SUBAPPLICATION Sitzventile (* Subapplication Type *)
  (* Standard: 61499-2 *)
  (* Version 1.0, 2023-02-11, franz *)
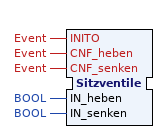
  EVENT_INPUT
    INITO;
    CNF_heben;
    CNF_senken;
  END_EVENT
  VAR_INPUT
    IN_heben : BOOL;
    IN_senken : BOOL;
  END_VAR
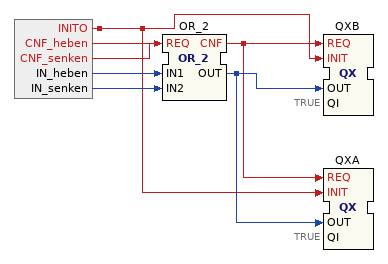
  FBS
    OR_2 : OR_2;
    QXB : QX(QI := TRUE);
    QXA : QX(QI := TRUE);
  END_FBS
  EVENT_CONNECTIONS
    OR_2.CNF TO QXB.REQ;
    OR_2.CNF TO QXA.REQ;
    CNF_heben TO OR_2.REQ;
    CNF_senken TO OR_2.REQ;
    INITO TO QXB.INIT;
    INITO TO QXA.INIT;
  END_CONNECTIONS
  DATA_CONNECTIONS
    OR_2.OUT TO QXB.OUT;
    OR_2.OUT TO QXA.OUT;
    IN_heben TO OR_2.IN1;
    IN_senken TO OR_2.IN2;
  END_CONNECTIONS
END_SUBAPPLICATION
